FUNCTION_BLOCK BACnetAnalogInput (* Service Interface Function Block Type *)
  (* Standard: 61499-2 *)
  (* Version 1.0, 2020-03-04, root *)
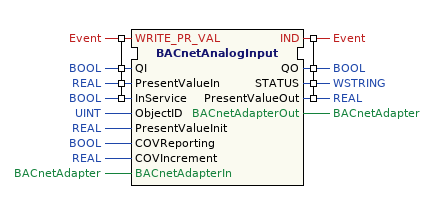
  EVENT_INPUT
    WRITE_PR_VAL WITH QI, PresentValueIn, InService; (* Write Present_Value event *)
  END_EVENT
  EVENT_OUTPUT
    IND WITH QO, STATUS, PresentValueOut; (* Present_Value write indication *)
  END_EVENT
  VAR_INPUT
    QI : BOOL; (* Event Input Qualifier *)
    PresentValueIn : REAL; (* Value to be written into the Present_Value property *)
    InService : BOOL; (* Lifestatus flag of the object *)
    ObjectID : UINT; (* Identifier of the object *)
    PresentValueInit : REAL; (* Initial value of the Present_Value property *)
    COVReporting : BOOL; (* Enable/Disable COV reporting flag *)
    COVIncrement : REAL; (* Difference in change required for triggering COV notifications *)
  END_VAR
  VAR_OUTPUT
    QO : BOOL; (* Event Output Qualifier *)
    STATUS : WSTRING; (* Status *)
    PresentValueOut : REAL; (* Value of the Present_Value property *)
  END_VAR
  SOCKETS
    BACnetAdapterIn : BACnetAdapter;
  END_SOCKETS
  PLUGS
    BACnetAdapterOut : BACnetAdapter; (* BACnet adapter plug *)
  END_PLUGS
END_FUNCTION_BLOCK
